INTERFACE PUBLIC I_MoveBuilder EXTENDS __System.IQueryInterface

METHOD PUBLIC Acceleration : I_MoveBuilder
VAR_INPUT
	value : LREAL;
END_VAR
END_METHOD

METHOD PUBLIC BufferMode : I_MoveBuilder
VAR_INPUT
	mode : AxisBufferMode;
END_VAR
END_METHOD

METHOD PUBLIC BuildMoveVelocityCommand : I_MoveCommand
END_METHOD

METHOD PUBLIC Deceleration : I_MoveBuilder
VAR_INPUT
	value : LREAL;
END_VAR
END_METHOD

METHOD PUBLIC Distance : I_MoveRelativeBuilder
VAR_INPUT
	value : LREAL;
END_VAR
END_METHOD

METHOD PUBLIC Jerk : I_MoveBuilder
VAR_INPUT
	value : LREAL;
END_VAR
END_METHOD

METHOD PUBLIC Position : I_MoveAbsoluteBuilder
VAR_INPUT
	value : LREAL;
END_VAR
END_METHOD

METHOD PUBLIC Velocity : I_MoveBuilder
VAR_INPUT
	value : LREAL;
END_VAR
END_METHOD

END_INTERFACE

(* stored: Version 1.1.0.1, ProductVersion 3.1.4024.12
   Itf I_MoveBuilder: Id {78b300c9-07ae-04a9-1036-4e6b5c3e54aa}
   Method Acceleration: Id {9ed5b283-467e-024e-1880-e4a5795709ff}
   Method BufferMode: Id {5df7c0f7-f9b3-075a-3997-a785fe25be8f}
   Method BuildMoveVelocityCommand: Id {7f51dcf0-37aa-06e9-2d7d-327b8a41a273}
   Method Deceleration: Id {d2747f03-3be5-0e18-3938-e6c0befd6f2b}
   Method Distance: Id {1daa1bfb-9cbc-05a2-22ad-de83d4f1fccf}
   Method Jerk: Id {3a3e9386-a52e-078c-1570-7aca32e96639}
   Method Position: Id {64e4fe0d-65bc-0f8b-0542-35b11001e6e1}
   Method Velocity: Id {80e14d95-4225-04d1-3482-772b10f531a1} *)
